FUNCTION F_ITC_SendMCR : BOOL
(**************************************************************************************
 * 	Application		:	BoxControl Framework
 *	Revision		:	$Revision: 404529 $
 *	Revision date	:	$Date: 2018-04-23 08:21:38 +0200 (Mo., 23 Apr 2018) $
 *	Last changed by	:	$Author: b7bolm $
 *	URL				:	$URL: http://almscdc.swisslog.com/repo/SWPD/Development/BoxControlFramework/20_Release/trunk/01_Software/BCF/BCF/JumpStart/20_Product/10_App/11_Com/10_Lib/10_Conv/11_ITC/F_ITC_SendMCR.TcPOU $
 *
 *	Purpose			:	Wrap message - MCR
 *
 * ------------------------------------------------------------------------------------
 *	Copyright Swisslog [IP AG], Switzerland. All rights reserved.
 * 
 * ------------------------------------------------------------------------------------
 *	
 * 	Revision History: 
 *
 * 	VERSION			DATE			INITIALS			DESCRIPTION
 *	0.1				01.01.2001		swl					Example
 *
 **************************************************************************************)
VAR_INPUT
	eChannelSrc			: E_MFCS_Channel; // Source communicaton channel	
	Position			: STRING(Conveyor.POSITION_STRINGLENGTH); // Position
	Code				: INT; // Code
	Mode				: INT; // Mode
	Speed				: ST_ITC_ManualMotionSpeed; // Speed
	Axis				: ARRAY[1..6] OF ST_ITC_ManualMotionAxis; // Axis
	Button				: ARRAY[1..2] OF ST_ITC_ManualMotionSelection; // Buttons
	eReturnCode			: E_ErrorConv; // Return code
END_VAR
VAR
	MCR					: ST_ITC_MCR; 
END_VAR

// Map values
MCR.Position := Position;
MCR.Speed := Speed;
MCR.Mode := Mode;
MCR.Code := Code;
MCR.Axis := Axis;
MCR.Button := Button;
MCR.eReturnCode := eReturnCode;

// Forward to ITC
F_ITC_SendMCR := fbITC_Manager.M_SendData(
					meChannel	:= eChannelSrc,
					mMsgType	:= E_ITC_MsgTypeConv.MANUAL_CONTROL_REPORT,
					mpData		:= ADR(MCR),
					mLen		:= SIZEOF(MCR));

END_FUNCTION

(* stored: Version 1.1.0.1, ProductVersion 3.1.4022.12
   POU F_ITC_SendMCR: Id {a2f7c278-fd92-4a04-9df7-24a1b091014f}, SpecialFunc None *)
